// TIA Portal V19 export
TYPE "AreaInterface"
// stored: Access Published
   STRUCT
      EStop : Bool;   // Machine Safe Stop Motion (Emergency Stop)
      Man : Bool;   // Machine Mode MANU
      Aut : Bool;   // Machine Mode AUTO
      Cycle : Bool;   // Machine CYCLE ON
      StopInPhase : Bool;   // Machine NORMAL CYCLE STOP
      StopProgrammed : Bool;   // Machine PROGRAMMED CYCLE STOP
      RstAlarms : Bool;   // Alarms reset command (need ACK)
      ManOneShot : Bool;   // Positive edge of Mode MANU
      AutOneShot : Bool;   // Positive edge of Mode AUTO
      CycleOneShot : Bool;   // Positive edge of CYCLE ON
      CheckAutReady : Bool;   // Check Machine in auto ready
   END_STRUCT;
END_TYPE
